% RSLogix 500 project STRAPPER 21-1-08 1220 - IN USE.RSS, saved by version 7.00.00.19 %
PROJECT "STRAPSYS"    % processor: MicroLogix 1500 %

PROGRAM FILES
  LAD 2 "MAIN"  17 rungs
  LAD 3 "INPUTS"  67 rungs
  LAD 4 "OUTPUTS"  55 rungs
  LAD 5 "INTERF OP"  16 rungs
  LAD 6 "COEFF."  16 rungs  % COEFFICIENT OF SEALING %
  LAD 7 "DISPENSER"  18 rungs
  LAD 8 "MH600"  137 rungs
  LAD 9 "ORGANIT."  67 rungs
  LAD 10 "PRESS"  78 rungs
  LAD 11 "PUSH_BUNK"  101 rungs
  LAD 12 "CHECKING"  10 rungs
  LAD 13 "INFEED"  25 rungs  % INFEED CONTROLS %
  LAD 14 "OUTFEED"  12 rungs  % OUTFEED CONTROLS %
  LAD 15 "RECIPES"  18 rungs  % PV RECIPE CONTROL %
  LAD 16 "ENCODER"  10 rungs  % ENCODER %
  LAD 17 "VSD"  10 rungs  % INFEED VSD'S %
  LAD 18 "RECIPE SEQ"  29 rungs

DATA FILES
  O0 OUTPUTS  9 elements
  I1 INPUT  10 elements
  S2 STATUS  66 elements
  B3 BINARY  30 elements
  T4 TIMER  52 elements
  C5 COUNTER  1 elements
  R6 CONTROL  1 elements
  N7 INTEGER  68 elements
  F8 FLOAT  9 elements
  N9 OP  13 elements
  B10 ORGANIT  106 elements
  N11 ON_SHOOT  3 elements
  L12   16 elements
  B20 MH600  101 elements
  B35 DISPENSER  9 elements
  B40 INFEEDBIN  100 elements  % INFEED SYSTEM BINARY %
  T41 INFEEDTIM  100 elements  % INFEED TIMERS %
  N42 INFEEDINT  100 elements  % INFEED INTEGERS %
  B50 PUSH_BUNK  24 elements
  N51 RECIPE  170 elements
  N52 REC NAMES  160 elements

LADDER 2 "MAIN"
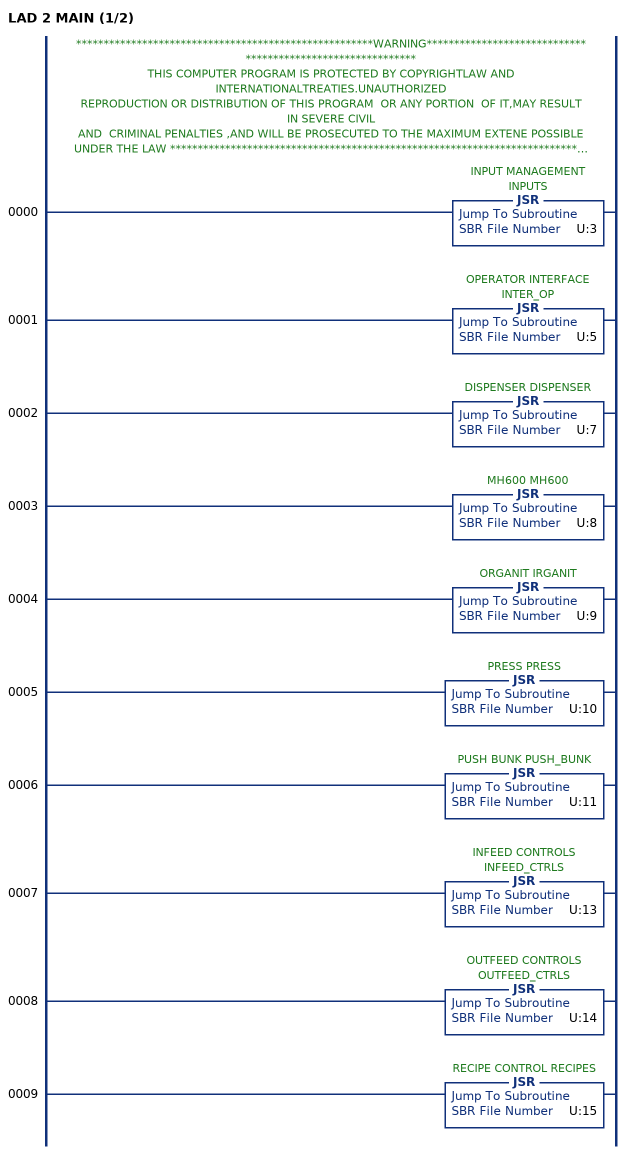
% Rung: 0 %
% ******************************************************WARNING************************************************************
% THIS COMPUTER PROGRAM IS PROTECTED BY COPYRIGHTLAW AND  INTERNATIONALTREATIES.UNAUTHORIZED
%  REPRODUCTION OR DISTRIBUTION OF THIS PROGRAM  OR ANY PORTION  OF IT,MAY RESULT IN SEVERE CIVIL
% AND  CRIMINAL PENALTIES ,AND WILL BE PROSECUTED TO THE MAXIMUM EXTENE POSSIBLE  UNDER THE LAW **************************************************************************************************************************
% Calls to the soubroutine %
SOR JSR U:3 EOR
%   U:3  INPUTS  "INPUT MANAGEMENT" %
% Rung: 1 %
SOR JSR U:5 EOR
%   U:5  INTER_OP  "OPERATOR INTERFACE" %
% Rung: 2 %
SOR JSR U:7 EOR
%   U:7  DISPENSER  "DISPENSER" %
% Rung: 3 %
SOR JSR U:8 EOR
%   U:8  MH600  "MH600" %
% Rung: 4 %
SOR JSR U:9 EOR
%   U:9  IRGANIT  "ORGANIT" %
% Rung: 5 %
SOR JSR U:10 EOR
%   U:10  PRESS  "PRESS" %
% Rung: 6 %
SOR JSR U:11 EOR
%   U:11  PUSH_BUNK  "PUSH BUNK" %
% Rung: 7 %
SOR JSR U:13 EOR
%   U:13  INFEED_CTRLS  "INFEED CONTROLS" %
% Rung: 8 %
SOR JSR U:14 EOR
%   U:14  OUTFEED_CTRLS  "OUTFEED CONTROLS" %
% Rung: 9 %
SOR JSR U:15 EOR
%   U:15  RECIPES  "RECIPE CONTROL" %

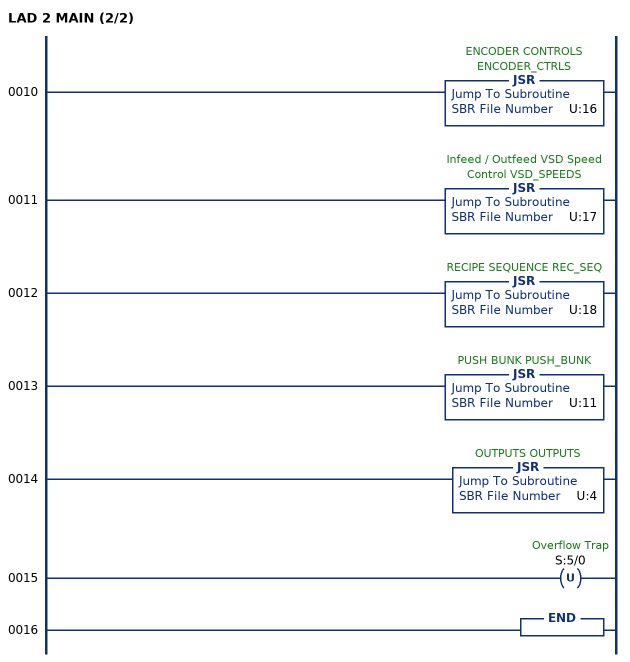
% Rung: 10 %
SOR JSR U:16 EOR
%   U:16  ENCODER_CTRLS  "ENCODER CONTROLS" %
% Rung: 11 %
SOR JSR U:17 EOR
%   U:17  VSD_SPEEDS  "Infeed / Outfeed VSD Speed Control" %
% Rung: 12 %
SOR JSR U:18 EOR
%   U:18  REC_SEQ  "RECIPE SEQUENCE" %
% Rung: 13 %
SOR JSR U:11 EOR
%   U:11  PUSH_BUNK  "PUSH BUNK" %
% Rung: 14 %
SOR JSR U:4 EOR
%   U:4  OUTPUTS  "OUTPUTS" %
% Rung: 15 %
SOR OTU S:5/0 EOR
%   S:5/0  "Overflow Trap" %
% Rung: 16 %
SOR END EOR

LADDER 3 "INPUTS"
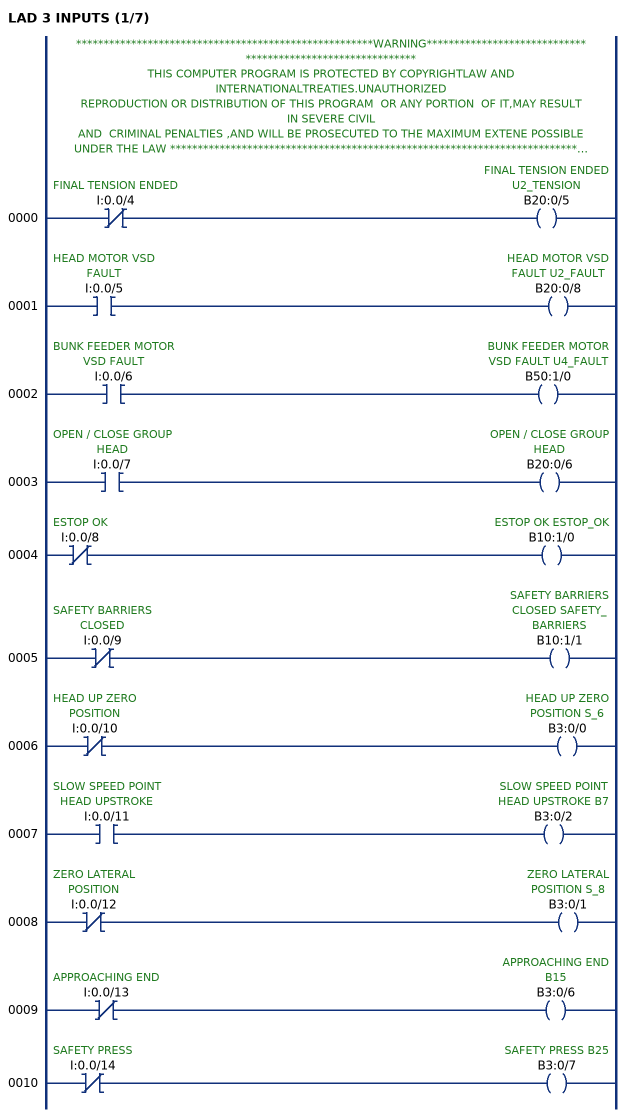
% Rung: 0 %
% ******************************************************WARNING************************************************************
% THIS COMPUTER PROGRAM IS PROTECTED BY COPYRIGHTLAW AND  INTERNATIONALTREATIES.UNAUTHORIZED
%  REPRODUCTION OR DISTRIBUTION OF THIS PROGRAM  OR ANY PORTION  OF IT,MAY RESULT IN SEVERE CIVIL
% AND  CRIMINAL PENALTIES ,AND WILL BE PROSECUTED TO THE MAXIMUM EXTENE POSSIBLE  UNDER THE LAW **************************************************************************************************************************
% AUTOMATIC VERTICAL PLASTIC MACHINE - I/O LOADING %
SOR XIO I:0.0/4 OTE B20:0/5 EOR
%   I:0.0/4  "FINAL TENSION ENDED" %
%   B20:0/5  U2_TENSION  "FINAL TENSION ENDED" %
% Rung: 1 %
SOR XIC I:0.0/5 OTE B20:0/8 EOR
%   I:0.0/5  "HEAD MOTOR VSD FAULT" %
%   B20:0/8  U2_FAULT  "HEAD MOTOR VSD FAULT" %
% Rung: 2 %
SOR XIC I:0.0/6 OTE B50:1/0 EOR
%   I:0.0/6  "BUNK FEEDER MOTOR VSD FAULT" %
%   B50:1/0  U4_FAULT  "BUNK FEEDER MOTOR VSD FAULT" %
% Rung: 3 %
SOR XIC I:0.0/7 OTE B20:0/6 EOR
%   I:0.0/7  "OPEN / CLOSE GROUP HEAD" %
%   B20:0/6  "OPEN / CLOSE GROUP HEAD" %
% Rung: 4 %
SOR XIO I:0.0/8 OTE B10:1/0 EOR
%   I:0.0/8  "ESTOP OK" %
%   B10:1/0  ESTOP_OK  "ESTOP OK" %
% Rung: 5 %
SOR XIO I:0.0/9 OTE B10:1/1 EOR
%   I:0.0/9  "SAFETY BARRIERS CLOSED" %
%   B10:1/1  SAFETY_BARRIERS  "SAFETY BARRIERS CLOSED" %
% Rung: 6 %
SOR XIO I:0.0/10 OTE B3:0/0 EOR
%   I:0.0/10  "HEAD UP ZERO POSITION" %
%   B3:0/0  S_6  "HEAD UP ZERO POSITION" %
% Rung: 7 %
SOR XIC I:0.0/11 OTE B3:0/2 EOR
%   I:0.0/11  "SLOW SPEED POINT HEAD UPSTROKE" %
%   B3:0/2  B7  "SLOW SPEED POINT HEAD UPSTROKE" %
% Rung: 8 %
SOR XIO I:0.0/12 OTE B3:0/1 EOR
%   I:0.0/12  "ZERO LATERAL POSITION" %
%   B3:0/1  S_8  "ZERO LATERAL POSITION" %
% Rung: 9 %
SOR XIO I:0.0/13 OTE B3:0/6 EOR
%   I:0.0/13  "APPROACHING END" %
%   B3:0/6  B15  "APPROACHING END" %
% Rung: 10 %
SOR XIO I:0.0/14 OTE B3:0/7 EOR
%   I:0.0/14  "SAFETY PRESS" %
%   B3:0/7  B25  "SAFETY PRESS" %

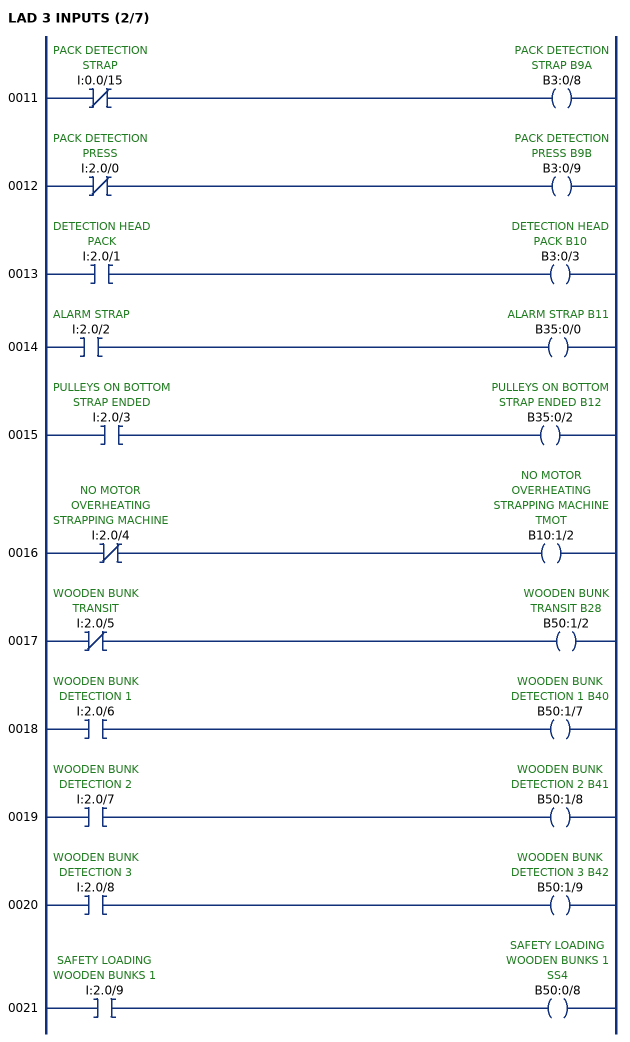
% Rung: 11 %
SOR XIO I:0.0/15 OTE B3:0/8 EOR
%   I:0.0/15  "PACK DETECTION STRAP" %
%   B3:0/8  B9A  "PACK DETECTION STRAP" %
% Rung: 12 %
SOR XIO I:2.0/0 OTE B3:0/9 EOR
%   I:2.0/0  "PACK DETECTION PRESS" %
%   B3:0/9  B9B  "PACK DETECTION PRESS" %
% Rung: 13 %
SOR XIC I:2.0/1 OTE B3:0/3 EOR
%   I:2.0/1  "DETECTION HEAD PACK" %
%   B3:0/3  B10  "DETECTION HEAD PACK" %
% Rung: 14 %
SOR XIC I:2.0/2 OTE B35:0/0 EOR
%   I:2.0/2  "ALARM STRAP" %
%   B35:0/0  B11  "ALARM STRAP" %
% Rung: 15 %
SOR XIC I:2.0/3 OTE B35:0/2 EOR
%   I:2.0/3  "PULLEYS ON BOTTOM STRAP ENDED" %
%   B35:0/2  B12  "PULLEYS ON BOTTOM STRAP ENDED" %
% Rung: 16 %
SOR XIO I:2.0/4 OTE B10:1/2 EOR
%   I:2.0/4  "NO MOTOR OVERHEATING STRAPPING MACHINE" %
%   B10:1/2  TMOT  "NO MOTOR OVERHEATING STRAPPING MACHINE" %
% Rung: 17 %
SOR XIO I:2.0/5 OTE B50:1/2 EOR
%   I:2.0/5  "WOODEN BUNK TRANSIT" %
%   B50:1/2  B28  "WOODEN BUNK TRANSIT" %
% Rung: 18 %
SOR XIC I:2.0/6 OTE B50:1/7 EOR
%   I:2.0/6  "WOODEN BUNK DETECTION 1" %
%   B50:1/7  B40  "WOODEN BUNK DETECTION 1" %
% Rung: 19 %
SOR XIC I:2.0/7 OTE B50:1/8 EOR
%   I:2.0/7  "WOODEN BUNK DETECTION 2" %
%   B50:1/8  B41  "WOODEN BUNK DETECTION 2" %
% Rung: 20 %
SOR XIC I:2.0/8 OTE B50:1/9 EOR
%   I:2.0/8  "WOODEN BUNK DETECTION 3" %
%   B50:1/9  B42  "WOODEN BUNK DETECTION 3" %
% Rung: 21 %
SOR XIC I:2.0/9 OTE B50:0/8 EOR
%   I:2.0/9  "SAFETY LOADING WOODEN BUNKS 1" %
%   B50:0/8  SS4  "SAFETY LOADING WOODEN BUNKS 1" %

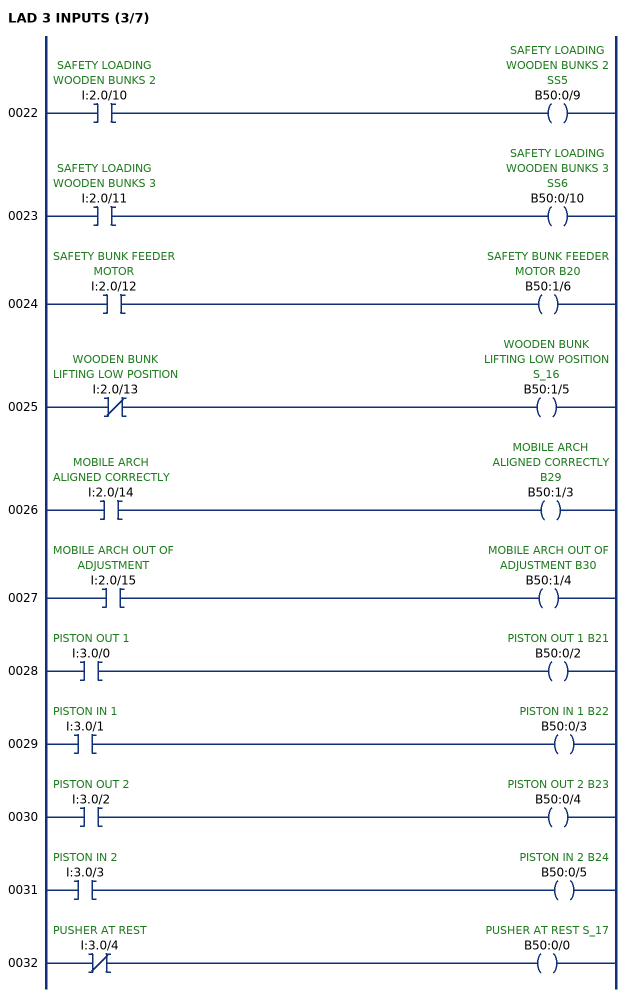
% Rung: 22 %
SOR XIC I:2.0/10 OTE B50:0/9 EOR
%   I:2.0/10  "SAFETY LOADING WOODEN BUNKS 2" %
%   B50:0/9  SS5  "SAFETY LOADING WOODEN BUNKS 2" %
% Rung: 23 %
SOR XIC I:2.0/11 OTE B50:0/10 EOR
%   I:2.0/11  "SAFETY LOADING WOODEN BUNKS 3" %
%   B50:0/10  SS6  "SAFETY LOADING WOODEN BUNKS 3" %
% Rung: 24 %
SOR XIC I:2.0/12 OTE B50:1/6 EOR
%   I:2.0/12  "SAFETY BUNK FEEDER MOTOR" %
%   B50:1/6  B20  "SAFETY BUNK FEEDER MOTOR" %
% Rung: 25 %
SOR XIO I:2.0/13 OTE B50:1/5 EOR
%   I:2.0/13  "WOODEN BUNK LIFTING LOW POSITION" %
%   B50:1/5  S_16  "WOODEN BUNK LIFTING LOW POSITION" %
% Rung: 26 %
SOR XIC I:2.0/14 OTE B50:1/3 EOR
%   I:2.0/14  "MOBILE ARCH ALIGNED CORRECTLY" %
%   B50:1/3  B29  "MOBILE ARCH ALIGNED CORRECTLY" %
% Rung: 27 %
SOR XIC I:2.0/15 OTE B50:1/4 EOR
%   I:2.0/15  "MOBILE ARCH OUT OF ADJUSTMENT" %
%   B50:1/4  B30  "MOBILE ARCH OUT OF ADJUSTMENT" %
% Rung: 28 %
SOR XIC I:3.0/0 OTE B50:0/2 EOR
%   I:3.0/0  "PISTON OUT 1" %
%   B50:0/2  B21  "PISTON OUT 1" %
% Rung: 29 %
SOR XIC I:3.0/1 OTE B50:0/3 EOR
%   I:3.0/1  "PISTON IN 1" %
%   B50:0/3  B22  "PISTON IN 1" %
% Rung: 30 %
SOR XIC I:3.0/2 OTE B50:0/4 EOR
%   I:3.0/2  "PISTON OUT 2" %
%   B50:0/4  B23  "PISTON OUT 2" %
% Rung: 31 %
SOR XIC I:3.0/3 OTE B50:0/5 EOR
%   I:3.0/3  "PISTON IN 2" %
%   B50:0/5  B24  "PISTON IN 2" %
% Rung: 32 %
SOR XIO I:3.0/4 OTE B50:0/0 EOR
%   I:3.0/4  "PUSHER AT REST" %
%   B50:0/0  S_17  "PUSHER AT REST" %

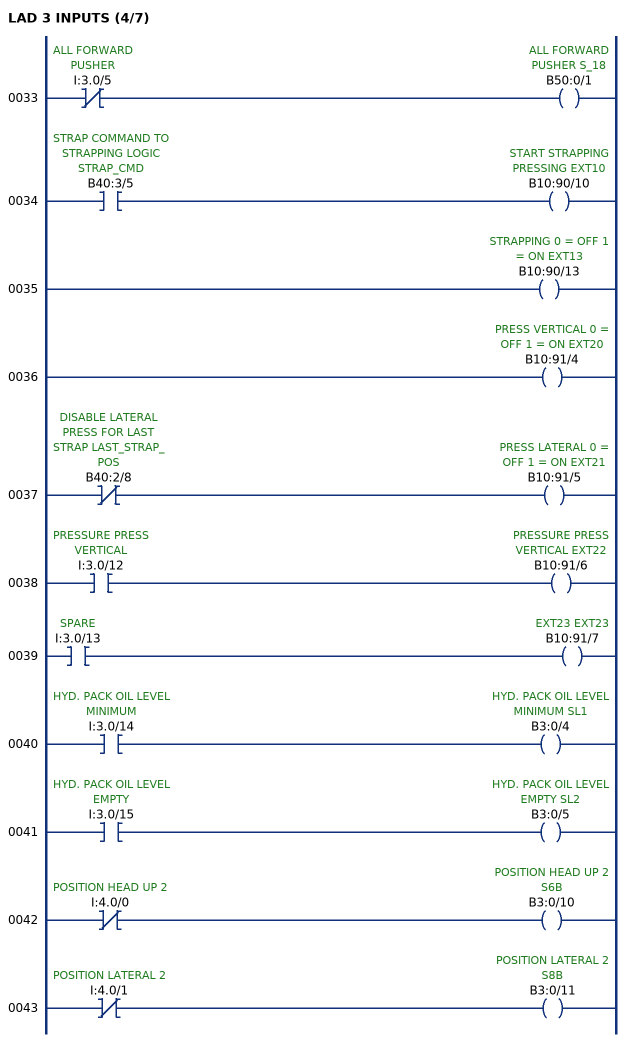
% Rung: 33 %
SOR XIO I:3.0/5 OTE B50:0/1 EOR
%   I:3.0/5  "ALL FORWARD PUSHER" %
%   B50:0/1  S_18  "ALL FORWARD PUSHER" %
% Rung: 34 %
SOR XIC B40:3/5 OTE B10:90/10 EOR
%   B40:3/5  STRAP_CMD  "STRAP COMMAND TO STRAPPING LOGIC" %
%   B10:90/10  EXT10  "START STRAPPING PRESSING" %
% Rung: 35 %
SOR OTE B10:90/13 EOR
%   B10:90/13  EXT13  "STRAPPING 0 = OFF 1 = ON" %
% Rung: 36 %
SOR OTE B10:91/4 EOR
%   B10:91/4  EXT20  "PRESS VERTICAL 0 = OFF 1 = ON" %
% Rung: 37 %
SOR XIO B40:2/8 OTE B10:91/5 EOR
%   B40:2/8  LAST_STRAP_POS  "DISABLE LATERAL PRESS FOR LAST STRAP" %
%   B10:91/5  EXT21  "PRESS LATERAL 0 = OFF 1 = ON" %
% Rung: 38 %
SOR XIC I:3.0/12 OTE B10:91/6 EOR
%   I:3.0/12  "PRESSURE PRESS VERTICAL" %
%   B10:91/6  EXT22  "PRESSURE PRESS VERTICAL" %
% Rung: 39 %
SOR XIC I:3.0/13 OTE B10:91/7 EOR
%   I:3.0/13  "SPARE" %
%   B10:91/7  EXT23  "EXT23" %
% Rung: 40 %
SOR XIC I:3.0/14 OTE B3:0/4 EOR
%   I:3.0/14  "HYD. PACK OIL LEVEL MINIMUM" %
%   B3:0/4  SL1  "HYD. PACK OIL LEVEL MINIMUM" %
% Rung: 41 %
SOR XIC I:3.0/15 OTE B3:0/5 EOR
%   I:3.0/15  "HYD. PACK OIL LEVEL EMPTY" %
%   B3:0/5  SL2  "HYD. PACK OIL LEVEL EMPTY" %
% Rung: 42 %
SOR XIO I:4.0/0 OTE B3:0/10 EOR
%   I:4.0/0  "POSITION HEAD UP 2" %
%   B3:0/10  S6B  "POSITION HEAD UP 2" %
% Rung: 43 %
SOR XIO I:4.0/1 OTE B3:0/11 EOR
%   I:4.0/1  "POSITION LATERAL 2" %
%   B3:0/11  S8B  "POSITION LATERAL 2" %

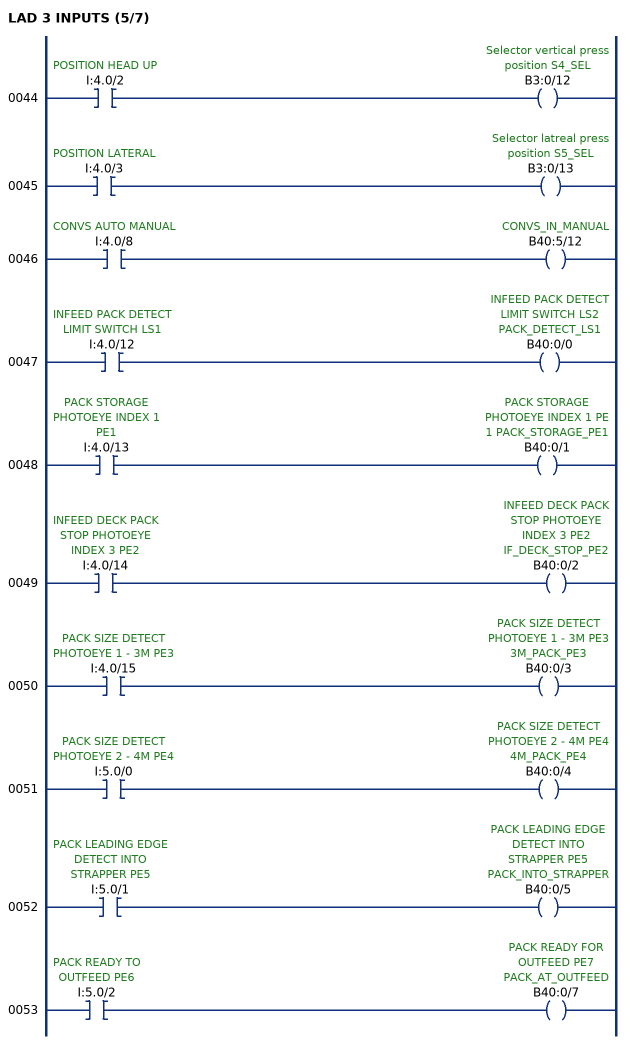
% Rung: 44 %
SOR XIC I:4.0/2 OTE B3:0/12 EOR
%   I:4.0/2  "POSITION HEAD UP" %
%   B3:0/12  S4_SEL  "Selector vertical press position" %
% Rung: 45 %
SOR XIC I:4.0/3 OTE B3:0/13 EOR
%   I:4.0/3  "POSITION LATERAL" %
%   B3:0/13  S5_SEL  "Selector latreal press position" %
% Rung: 46 %
SOR XIC I:4.0/8 OTE B40:5/12 EOR
%   I:4.0/8  "CONVS AUTO MANUAL" %
%   B40:5/12  CONVS_IN_MANUAL %
% Rung: 47 %
SOR XIC I:4.0/12 OTE B40:0/0 EOR
%   I:4.0/12  "INFEED PACK DETECT LIMIT SWITCH LS1" %
%   B40:0/0  PACK_DETECT_LS1  "INFEED PACK DETECT LIMIT SWITCH LS2" %
% Rung: 48 %
SOR XIC I:4.0/13 OTE B40:0/1 EOR
%   I:4.0/13  "PACK STORAGE PHOTOEYE INDEX 1 PE1" %
%   B40:0/1  PACK_STORAGE_PE1  "PACK STORAGE PHOTOEYE INDEX 1 PE 1" %
% Rung: 49 %
SOR XIC I:4.0/14 OTE B40:0/2 EOR
%   I:4.0/14  "INFEED DECK PACK STOP PHOTOEYE INDEX 3 PE2" %
%   B40:0/2  IF_DECK_STOP_PE2  "INFEED DECK PACK STOP PHOTOEYE INDEX 3 PE2" %
% Rung: 50 %
SOR XIC I:4.0/15 OTE B40:0/3 EOR
%   I:4.0/15  "PACK SIZE DETECT PHOTOEYE 1 - 3M PE3" %
%   B40:0/3  3M_PACK_PE3  "PACK SIZE DETECT PHOTOEYE 1 - 3M PE3" %
% Rung: 51 %
SOR XIC I:5.0/0 OTE B40:0/4 EOR
%   I:5.0/0  "PACK SIZE DETECT PHOTOEYE 2 - 4M PE4" %
%   B40:0/4  4M_PACK_PE4  "PACK SIZE DETECT PHOTOEYE 2 - 4M PE4" %
% Rung: 52 %
SOR XIC I:5.0/1 OTE B40:0/5 EOR
%   I:5.0/1  "PACK LEADING EDGE DETECT INTO STRAPPER PE5" %
%   B40:0/5  PACK_INTO_STRAPPER  "PACK LEADING EDGE DETECT INTO STRAPPER PE5" %
% Rung: 53 %
SOR XIC I:5.0/2 OTE B40:0/7 EOR
%   I:5.0/2  "PACK READY TO OUTFEED PE6" %
%   B40:0/7  PACK_AT_OUTFEED  "PACK READY FOR OUTFEED PE7" %

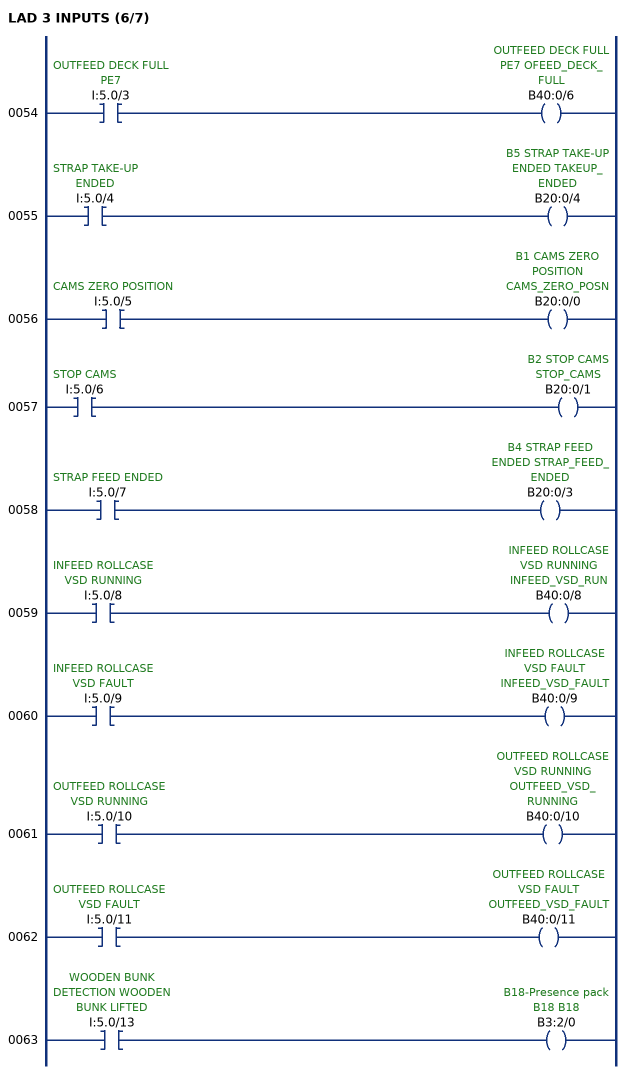
% Rung: 54 %
SOR XIC I:5.0/3 OTE B40:0/6 EOR
%   I:5.0/3  "OUTFEED DECK FULL PE7" %
%   B40:0/6  OFEED_DECK_FULL  "OUTFEED DECK FULL PE7" %
% Rung: 55 %
SOR XIC I:5.0/4 OTE B20:0/4 EOR
%   I:5.0/4  "STRAP TAKE-UP ENDED" %
%   B20:0/4  TAKEUP_ENDED  "B5 STRAP TAKE-UP ENDED" %
% Rung: 56 %
SOR XIC I:5.0/5 OTE B20:0/0 EOR
%   I:5.0/5  "CAMS ZERO POSITION" %
%   B20:0/0  CAMS_ZERO_POSN  "B1 CAMS ZERO POSITION" %
% Rung: 57 %
SOR XIC I:5.0/6 OTE B20:0/1 EOR
%   I:5.0/6  "STOP CAMS" %
%   B20:0/1  STOP_CAMS  "B2 STOP CAMS" %
% Rung: 58 %
SOR XIC I:5.0/7 OTE B20:0/3 EOR
%   I:5.0/7  "STRAP FEED ENDED" %
%   B20:0/3  STRAP_FEED_ENDED  "B4 STRAP FEED ENDED" %
% Rung: 59 %
SOR XIC I:5.0/8 OTE B40:0/8 EOR
%   I:5.0/8  "INFEED ROLLCASE VSD RUNNING" %
%   B40:0/8  INFEED_VSD_RUN  "INFEED ROLLCASE VSD RUNNING" %
% Rung: 60 %
SOR XIC I:5.0/9 OTE B40:0/9 EOR
%   I:5.0/9  "INFEED ROLLCASE VSD FAULT" %
%   B40:0/9  INFEED_VSD_FAULT  "INFEED ROLLCASE VSD FAULT" %
% Rung: 61 %
SOR XIC I:5.0/10 OTE B40:0/10 EOR
%   I:5.0/10  "OUTFEED ROLLCASE VSD RUNNING" %
%   B40:0/10  OUTFEED_VSD_RUNNING  "OUTFEED ROLLCASE VSD RUNNING" %
% Rung: 62 %
SOR XIC I:5.0/11 OTE B40:0/11 EOR
%   I:5.0/11  "OUTFEED ROLLCASE VSD FAULT" %
%   B40:0/11  OUTFEED_VSD_FAULT  "OUTFEED ROLLCASE VSD FAULT" %
% Rung: 63 %
SOR XIC I:5.0/13 OTE B3:2/0 EOR
%   I:5.0/13  "WOODEN BUNK DETECTION WOODEN BUNK LIFTED" %
%   B3:2/0  B18  "B18-Presence pack B18" %

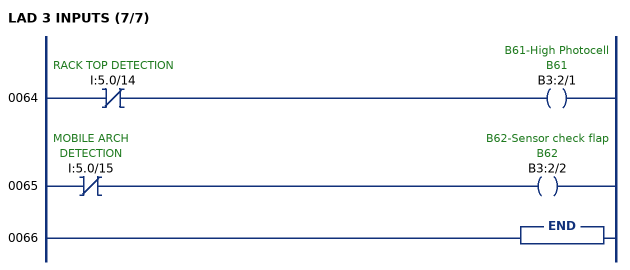
% Rung: 64 %
SOR XIO I:5.0/14 OTE B3:2/1 EOR
%   I:5.0/14  "RACK TOP DETECTION" %
%   B3:2/1  B61  "B61-High Photocell" %
% Rung: 65 %
SOR XIO I:5.0/15 OTE B3:2/2 EOR
%   I:5.0/15  "MOBILE ARCH DETECTION" %
%   B3:2/2  B62  "B62-Sensor check flap" %
% Rung: 66 %
SOR END EOR

LADDER 4 "OUTPUTS"
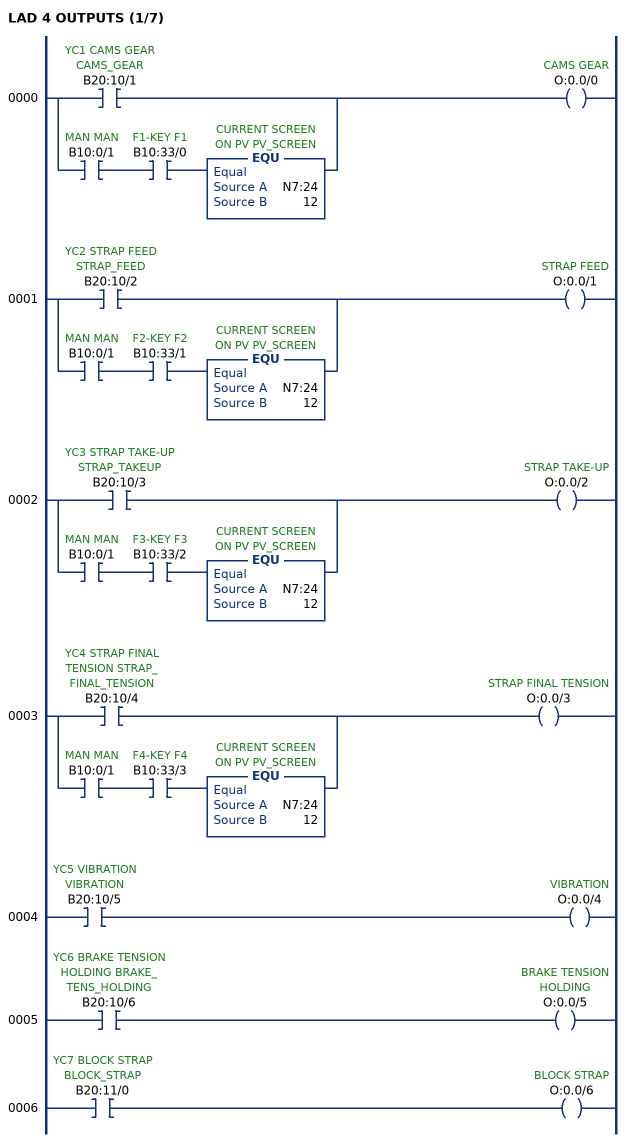
% Rung: 0 %
SOR BST XIC B20:10/1 NXB XIC B10:0/1 XIC B10:33/0 EQU N7:24 12 BND OTE O:0.0/0 EOR
%   B20:10/1  CAMS_GEAR  "YC1 CAMS GEAR" %
%   B10:0/1  MAN  "MAN" %
%   B10:33/0  F1  "F1-KEY" %
%   N7:24  PV_SCREEN  "CURRENT SCREEN ON PV" %
%   O:0.0/0  "CAMS GEAR" %
% Rung: 1 %
SOR BST XIC B20:10/2 NXB XIC B10:0/1 XIC B10:33/1 EQU N7:24 12 BND OTE O:0.0/1 EOR
%   B20:10/2  STRAP_FEED  "YC2 STRAP FEED" %
%   B10:0/1  MAN  "MAN" %
%   B10:33/1  F2  "F2-KEY" %
%   N7:24  PV_SCREEN  "CURRENT SCREEN ON PV" %
%   O:0.0/1  "STRAP FEED" %
% Rung: 2 %
SOR BST XIC B20:10/3 NXB XIC B10:0/1 XIC B10:33/2 EQU N7:24 12 BND OTE O:0.0/2 EOR
%   B20:10/3  STRAP_TAKEUP  "YC3 STRAP TAKE-UP" %
%   B10:0/1  MAN  "MAN" %
%   B10:33/2  F3  "F3-KEY" %
%   N7:24  PV_SCREEN  "CURRENT SCREEN ON PV" %
%   O:0.0/2  "STRAP TAKE-UP" %
% Rung: 3 %
SOR BST XIC B20:10/4 NXB XIC B10:0/1 XIC B10:33/3 EQU N7:24 12 BND OTE O:0.0/3 EOR
%   B20:10/4  STRAP_FINAL_TENSION  "YC4 STRAP FINAL TENSION" %
%   B10:0/1  MAN  "MAN" %
%   B10:33/3  F4  "F4-KEY" %
%   N7:24  PV_SCREEN  "CURRENT SCREEN ON PV" %
%   O:0.0/3  "STRAP FINAL TENSION" %
% Rung: 4 %
SOR XIC B20:10/5 OTE O:0.0/4 EOR
%   B20:10/5  VIBRATION  "YC5 VIBRATION" %
%   O:0.0/4  "VIBRATION" %
% Rung: 5 %
SOR XIC B20:10/6 OTE O:0.0/5 EOR
%   B20:10/6  BRAKE_TENS_HOLDING  "YC6 BRAKE TENSION HOLDING" %
%   O:0.0/5  "BRAKE TENSION HOLDING" %
% Rung: 6 %
SOR XIC B20:11/0 OTE O:0.0/6 EOR
%   B20:11/0  BLOCK_STRAP  "YC7 BLOCK STRAP" %
%   O:0.0/6  "BLOCK STRAP" %

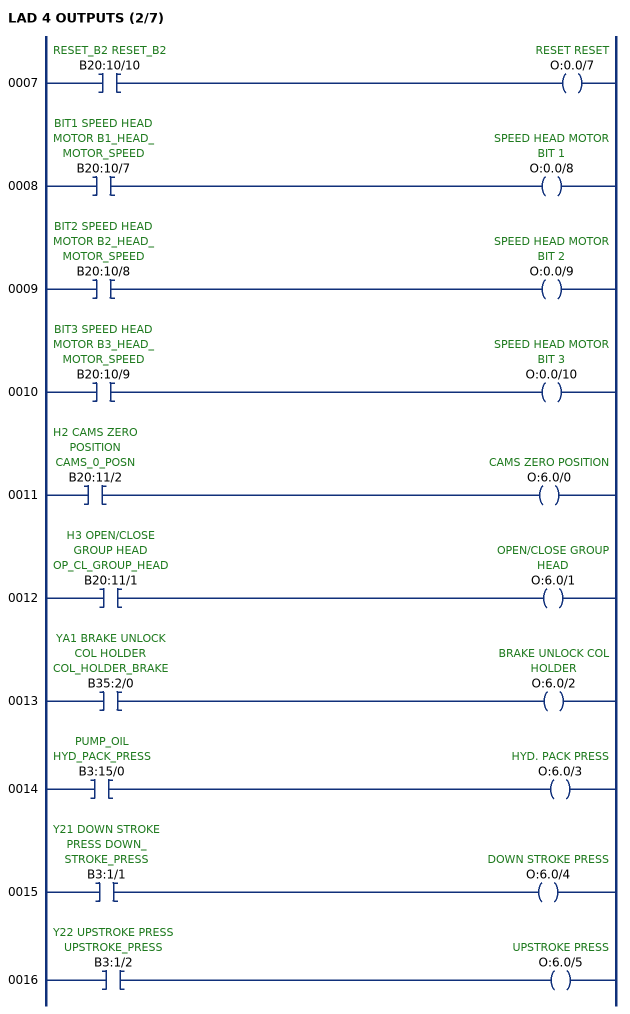
% Rung: 7 %
SOR XIC B20:10/10 OTE O:0.0/7 EOR
%   B20:10/10  RESET_B2  "RESET_B2" %
%   O:0.0/7  RESET  "RESET" %
% Rung: 8 %
SOR XIC B20:10/7 OTE O:0.0/8 EOR
%   B20:10/7  B1_HEAD_MOTOR_SPEED  "BIT1 SPEED HEAD MOTOR" %
%   O:0.0/8  "SPEED HEAD MOTOR BIT 1" %
% Rung: 9 %
SOR XIC B20:10/8 OTE O:0.0/9 EOR
%   B20:10/8  B2_HEAD_MOTOR_SPEED  "BIT2 SPEED HEAD MOTOR" %
%   O:0.0/9  "SPEED HEAD MOTOR BIT 2" %
% Rung: 10 %
SOR XIC B20:10/9 OTE O:0.0/10 EOR
%   B20:10/9  B3_HEAD_MOTOR_SPEED  "BIT3 SPEED HEAD MOTOR" %
%   O:0.0/10  "SPEED HEAD MOTOR BIT 3" %
% Rung: 11 %
SOR XIC B20:11/2 OTE O:6.0/0 EOR
%   B20:11/2  CAMS_0_POSN  "H2 CAMS ZERO POSITION" %
%   O:6.0/0  "CAMS ZERO POSITION" %
% Rung: 12 %
SOR XIC B20:11/1 OTE O:6.0/1 EOR
%   B20:11/1  OP_CL_GROUP_HEAD  "H3 OPEN/CLOSE GROUP HEAD" %
%   O:6.0/1  "OPEN/CLOSE GROUP HEAD" %
% Rung: 13 %
SOR XIC B35:2/0 OTE O:6.0/2 EOR
%   B35:2/0  COL_HOLDER_BRAKE  "YA1 BRAKE UNLOCK COL HOLDER" %
%   O:6.0/2  "BRAKE UNLOCK COL HOLDER" %
% Rung: 14 %
SOR XIC B3:15/0 OTE O:6.0/3 EOR
%   B3:15/0  HYD_PACK_PRESS  "PUMP_OIL" %
%   O:6.0/3  "HYD. PACK PRESS" %
% Rung: 15 %
SOR XIC B3:1/1 OTE O:6.0/4 EOR
%   B3:1/1  DOWN_STROKE_PRESS  "Y21 DOWN STROKE PRESS" %
%   O:6.0/4  "DOWN STROKE PRESS" %
% Rung: 16 %
SOR XIC B3:1/2 OTE O:6.0/5 EOR
%   B3:1/2  UPSTROKE_PRESS  "Y22 UPSTROKE PRESS" %
%   O:6.0/5  "UPSTROKE PRESS" %

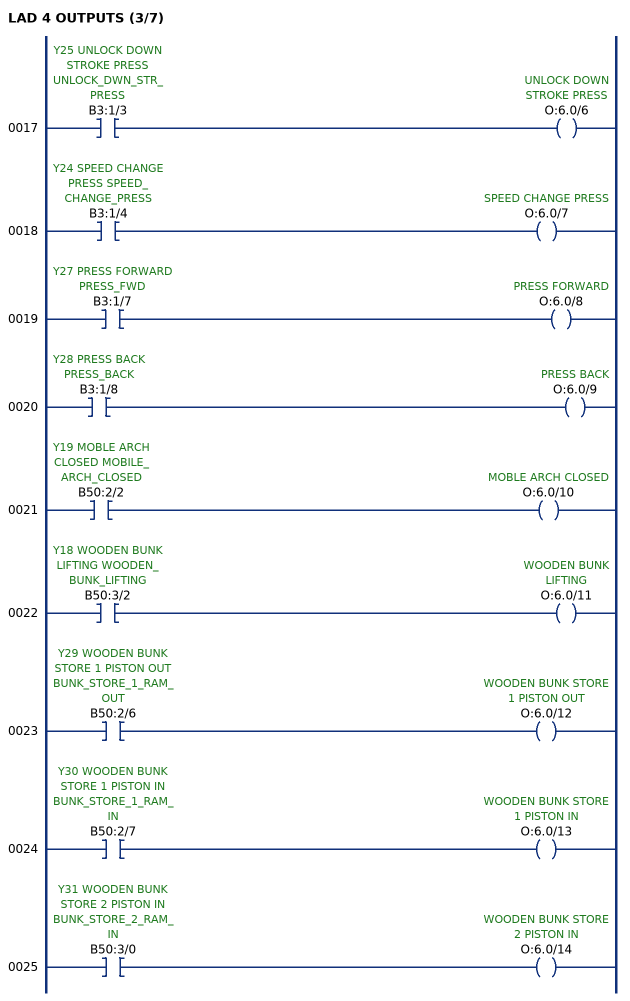
% Rung: 17 %
SOR XIC B3:1/3 OTE O:6.0/6 EOR
%   B3:1/3  UNLOCK_DWN_STR_PRESS  "Y25 UNLOCK DOWN STROKE PRESS" %
%   O:6.0/6  "UNLOCK DOWN STROKE PRESS" %
% Rung: 18 %
SOR XIC B3:1/4 OTE O:6.0/7 EOR
%   B3:1/4  SPEED_CHANGE_PRESS  "Y24 SPEED CHANGE PRESS" %
%   O:6.0/7  "SPEED CHANGE PRESS" %
% Rung: 19 %
SOR XIC B3:1/7 OTE O:6.0/8 EOR
%   B3:1/7  PRESS_FWD  "Y27 PRESS FORWARD" %
%   O:6.0/8  "PRESS FORWARD" %
% Rung: 20 %
SOR XIC B3:1/8 OTE O:6.0/9 EOR
%   B3:1/8  PRESS_BACK  "Y28 PRESS BACK" %
%   O:6.0/9  "PRESS BACK" %
% Rung: 21 %
SOR XIC B50:2/2 OTE O:6.0/10 EOR
%   B50:2/2  MOBILE_ARCH_CLOSED  "Y19 MOBLE ARCH CLOSED" %
%   O:6.0/10  "MOBLE ARCH CLOSED" %
% Rung: 22 %
SOR XIC B50:3/2 OTE O:6.0/11 EOR
%   B50:3/2  WOODEN_BUNK_LIFTING  "Y18 WOODEN BUNK LIFTING" %
%   O:6.0/11  "WOODEN BUNK LIFTING" %
% Rung: 23 %
SOR XIC B50:2/6 OTE O:6.0/12 EOR
%   B50:2/6  BUNK_STORE_1_RAM_OUT  "Y29 WOODEN BUNK STORE 1 PISTON OUT" %
%   O:6.0/12  "WOODEN BUNK STORE 1 PISTON OUT" %
% Rung: 24 %
SOR XIC B50:2/7 OTE O:6.0/13 EOR
%   B50:2/7  BUNK_STORE_1_RAM_IN  "Y30 WOODEN BUNK STORE 1 PISTON IN" %
%   O:6.0/13  "WOODEN BUNK STORE 1 PISTON IN" %
% Rung: 25 %
SOR XIC B50:3/0 OTE O:6.0/14 EOR
%   B50:3/0  BUNK_STORE_2_RAM_IN  "Y31 WOODEN BUNK STORE 2 PISTON IN" %
%   O:6.0/14  "WOODEN BUNK STORE 2 PISTON IN" %

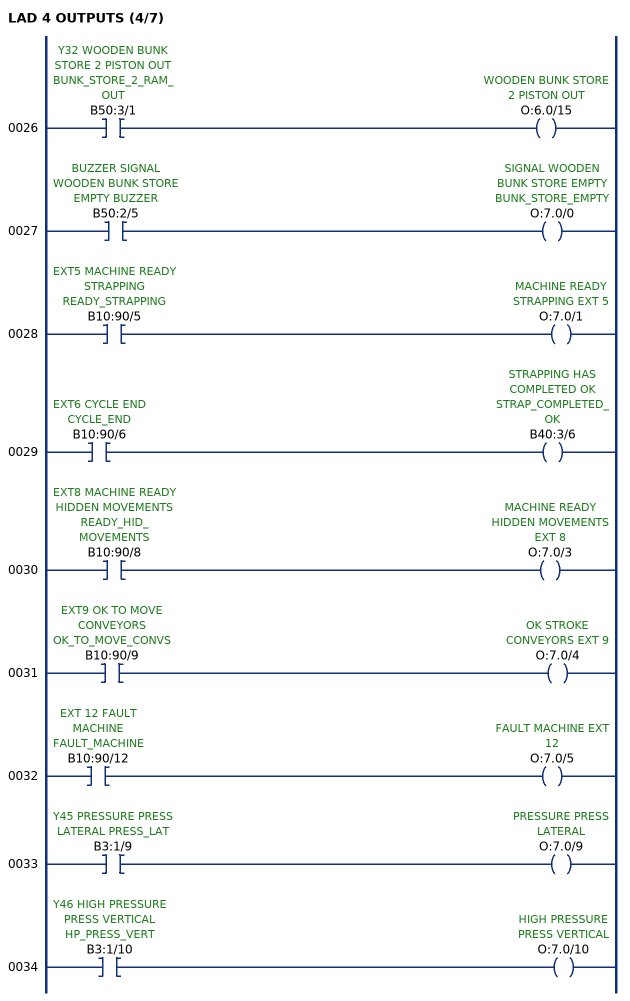
% Rung: 26 %
SOR XIC B50:3/1 OTE O:6.0/15 EOR
%   B50:3/1  BUNK_STORE_2_RAM_OUT  "Y32 WOODEN BUNK STORE 2 PISTON OUT" %
%   O:6.0/15  "WOODEN BUNK STORE 2 PISTON OUT" %
% Rung: 27 %
SOR XIC B50:2/5 OTE O:7.0/0 EOR
%   B50:2/5  BUZZER  "BUZZER SIGNAL WOODEN BUNK STORE EMPTY" %
%   O:7.0/0  BUNK_STORE_EMPTY  "SIGNAL WOODEN BUNK STORE EMPTY" %
% Rung: 28 %
SOR XIC B10:90/5 OTE O:7.0/1 EOR
%   B10:90/5  READY_STRAPPING  "EXT5 MACHINE READY STRAPPING" %
%   O:7.0/1  "MACHINE READY STRAPPING EXT 5" %
% Rung: 29 %
SOR XIC B10:90/6 OTE B40:3/6 EOR
%   B10:90/6  CYCLE_END  "EXT6 CYCLE END" %
%   B40:3/6  STRAP_COMPLETED_OK  "STRAPPING HAS COMPLETED OK" %
% Rung: 30 %
SOR XIC B10:90/8 OTE O:7.0/3 EOR
%   B10:90/8  READY_HID_MOVEMENTS  "EXT8 MACHINE READY HIDDEN MOVEMENTS" %
%   O:7.0/3  "MACHINE READY HIDDEN MOVEMENTS EXT 8" %
% Rung: 31 %
SOR XIC B10:90/9 OTE O:7.0/4 EOR
%   B10:90/9  OK_TO_MOVE_CONVS  "EXT9 OK TO MOVE CONVEYORS" %
%   O:7.0/4  "OK STROKE CONVEYORS EXT 9" %
% Rung: 32 %
SOR XIC B10:90/12 OTE O:7.0/5 EOR
%   B10:90/12  FAULT_MACHINE  "EXT 12 FAULT MACHINE" %
%   O:7.0/5  "FAULT MACHINE EXT 12" %
% Rung: 33 %
SOR XIC B3:1/9 OTE O:7.0/9 EOR
%   B3:1/9  PRESS_LAT  "Y45 PRESSURE PRESS LATERAL" %
%   O:7.0/9  "PRESSURE PRESS LATERAL" %
% Rung: 34 %
SOR XIC B3:1/10 OTE O:7.0/10 EOR
%   B3:1/10  HP_PRESS_VERT  "Y46 HIGH PRESSURE PRESS VERTICAL" %
%   O:7.0/10  "HIGH PRESSURE PRESS VERTICAL" %

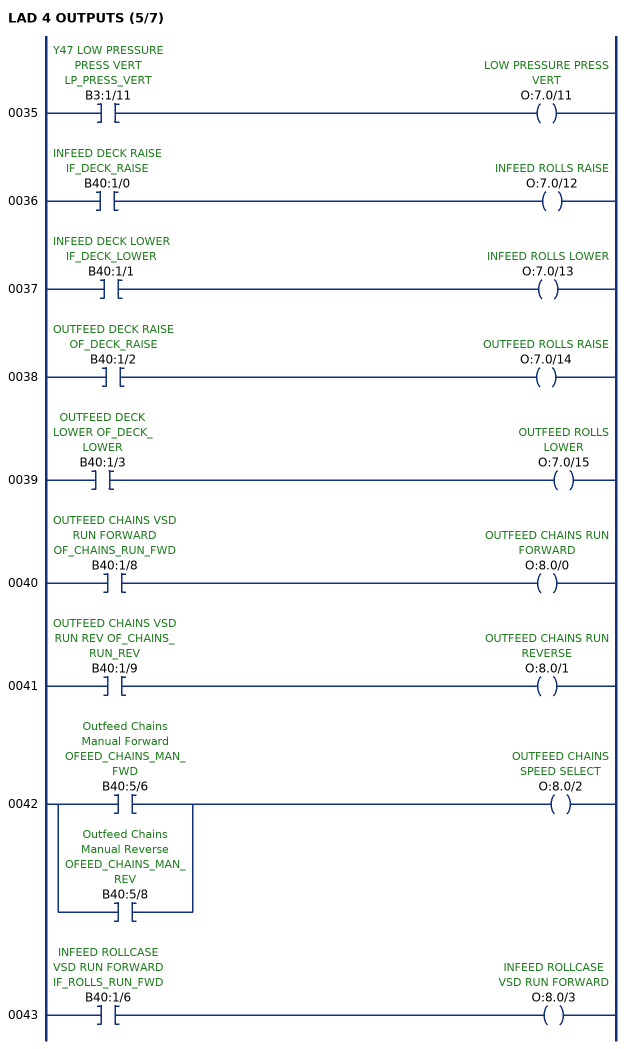
% Rung: 35 %
SOR XIC B3:1/11 OTE O:7.0/11 EOR
%   B3:1/11  LP_PRESS_VERT  "Y47 LOW PRESSURE PRESS VERT" %
%   O:7.0/11  "LOW PRESSURE PRESS VERT" %
% Rung: 36 %
SOR XIC B40:1/0 OTE O:7.0/12 EOR
%   B40:1/0  IF_DECK_RAISE  "INFEED DECK RAISE" %
%   O:7.0/12  "INFEED ROLLS RAISE" %
% Rung: 37 %
SOR XIC B40:1/1 OTE O:7.0/13 EOR
%   B40:1/1  IF_DECK_LOWER  "INFEED DECK LOWER" %
%   O:7.0/13  "INFEED ROLLS LOWER" %
% Rung: 38 %
SOR XIC B40:1/2 OTE O:7.0/14 EOR
%   B40:1/2  OF_DECK_RAISE  "OUTFEED DECK RAISE" %
%   O:7.0/14  "OUTFEED ROLLS RAISE" %
% Rung: 39 %
SOR XIC B40:1/3 OTE O:7.0/15 EOR
%   B40:1/3  OF_DECK_LOWER  "OUTFEED DECK LOWER" %
%   O:7.0/15  "OUTFEED ROLLS LOWER" %
% Rung: 40 %
SOR XIC B40:1/8 OTE O:8.0/0 EOR
%   B40:1/8  OF_CHAINS_RUN_FWD  "OUTFEED CHAINS VSD RUN FORWARD" %
%   O:8.0/0  "OUTFEED CHAINS RUN FORWARD" %
% Rung: 41 %
SOR XIC B40:1/9 OTE O:8.0/1 EOR
%   B40:1/9  OF_CHAINS_RUN_REV  "OUTFEED CHAINS VSD RUN REV" %
%   O:8.0/1  "OUTFEED CHAINS RUN REVERSE" %
% Rung: 42 %
SOR BST XIC B40:5/6 NXB XIC B40:5/8 BND OTE O:8.0/2 EOR
%   B40:5/6  OFEED_CHAINS_MAN_FWD  "Outfeed Chains Manual Forward" %
%   B40:5/8  OFEED_CHAINS_MAN_REV  "Outfeed Chains Manual Reverse" %
%   O:8.0/2  "OUTFEED CHAINS SPEED SELECT" %
% Rung: 43 %
SOR XIC B40:1/6 OTE O:8.0/3 EOR
%   B40:1/6  IF_ROLLS_RUN_FWD  "INFEED ROLLCASE VSD RUN FORWARD" %
%   O:8.0/3  "INFEED ROLLCASE VSD RUN FORWARD" %

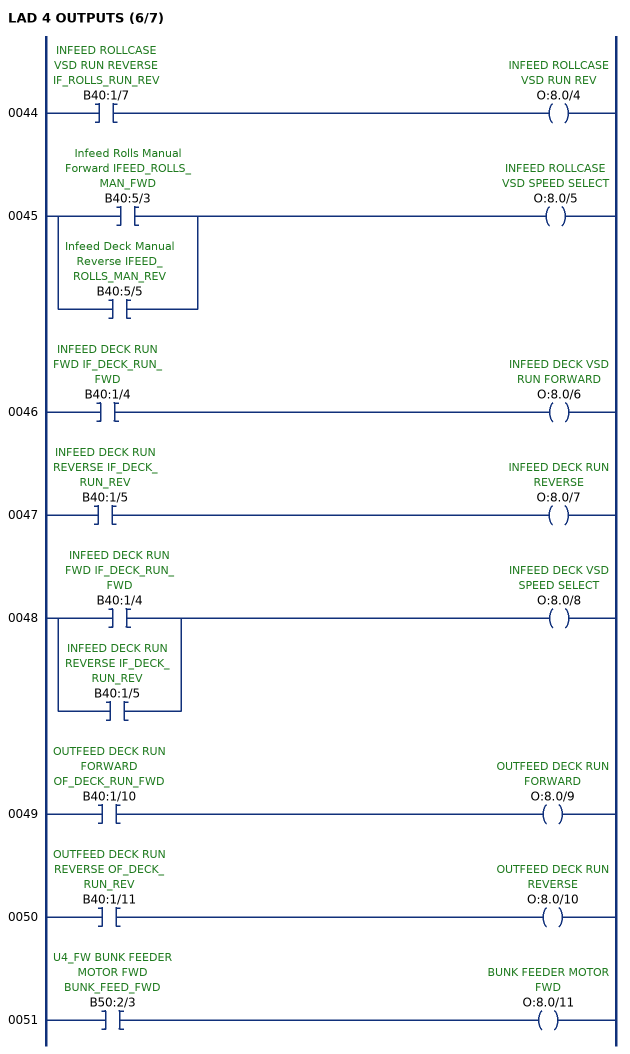
% Rung: 44 %
SOR XIC B40:1/7 OTE O:8.0/4 EOR
%   B40:1/7  IF_ROLLS_RUN_REV  "INFEED ROLLCASE VSD RUN REVERSE" %
%   O:8.0/4  "INFEED ROLLCASE VSD RUN REV" %
% Rung: 45 %
SOR BST XIC B40:5/3 NXB XIC B40:5/5 BND OTE O:8.0/5 EOR
%   B40:5/3  IFEED_ROLLS_MAN_FWD  "Infeed Rolls Manual Forward" %
%   B40:5/5  IFEED_ROLLS_MAN_REV  "Infeed Deck Manual Reverse" %
%   O:8.0/5  "INFEED ROLLCASE VSD SPEED SELECT" %
% Rung: 46 %
SOR XIC B40:1/4 OTE O:8.0/6 EOR
%   B40:1/4  IF_DECK_RUN_FWD  "INFEED DECK RUN FWD" %
%   O:8.0/6  "INFEED DECK VSD RUN FORWARD" %
% Rung: 47 %
SOR XIC B40:1/5 OTE O:8.0/7 EOR
%   B40:1/5  IF_DECK_RUN_REV  "INFEED DECK RUN REVERSE" %
%   O:8.0/7  "INFEED DECK RUN REVERSE" %
% Rung: 48 %
SOR BST XIC B40:1/4 NXB XIC B40:1/5 BND OTE O:8.0/8 EOR
%   B40:1/4  IF_DECK_RUN_FWD  "INFEED DECK RUN FWD" %
%   B40:1/5  IF_DECK_RUN_REV  "INFEED DECK RUN REVERSE" %
%   O:8.0/8  "INFEED DECK VSD SPEED SELECT" %
% Rung: 49 %
SOR XIC B40:1/10 OTE O:8.0/9 EOR
%   B40:1/10  OF_DECK_RUN_FWD  "OUTFEED DECK RUN FORWARD" %
%   O:8.0/9  "OUTFEED DECK RUN FORWARD" %
% Rung: 50 %
SOR XIC B40:1/11 OTE O:8.0/10 EOR
%   B40:1/11  OF_DECK_RUN_REV  "OUTFEED DECK RUN REVERSE" %
%   O:8.0/10  "OUTFEED DECK RUN REVERSE" %
% Rung: 51 %
SOR XIC B50:2/3 OTE O:8.0/11 EOR
%   B50:2/3  BUNK_FEED_FWD  "U4_FW BUNK FEEDER MOTOR FWD" %
%   O:8.0/11  "BUNK FEEDER MOTOR FWD" %

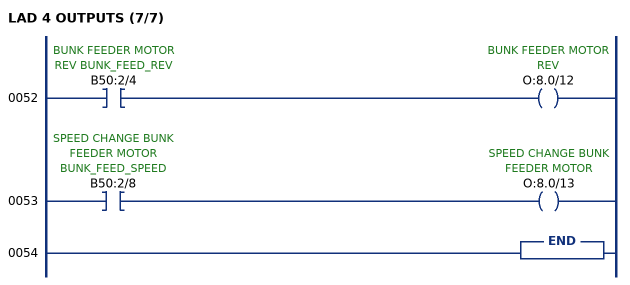
% Rung: 52 %
SOR XIC B50:2/4 OTE O:8.0/12 EOR
%   B50:2/4  BUNK_FEED_REV  "BUNK FEEDER MOTOR REV" %
%   O:8.0/12  "BUNK FEEDER MOTOR REV" %
% Rung: 53 %
SOR XIC B50:2/8 OTE O:8.0/13 EOR
%   B50:2/8  BUNK_FEED_SPEED  "SPEED CHANGE BUNK FEEDER MOTOR" %
%   O:8.0/13  "SPEED CHANGE BUNK FEEDER MOTOR" %
% Rung: 54 %
SOR END EOR

LADDER 5 "INTERF OP"
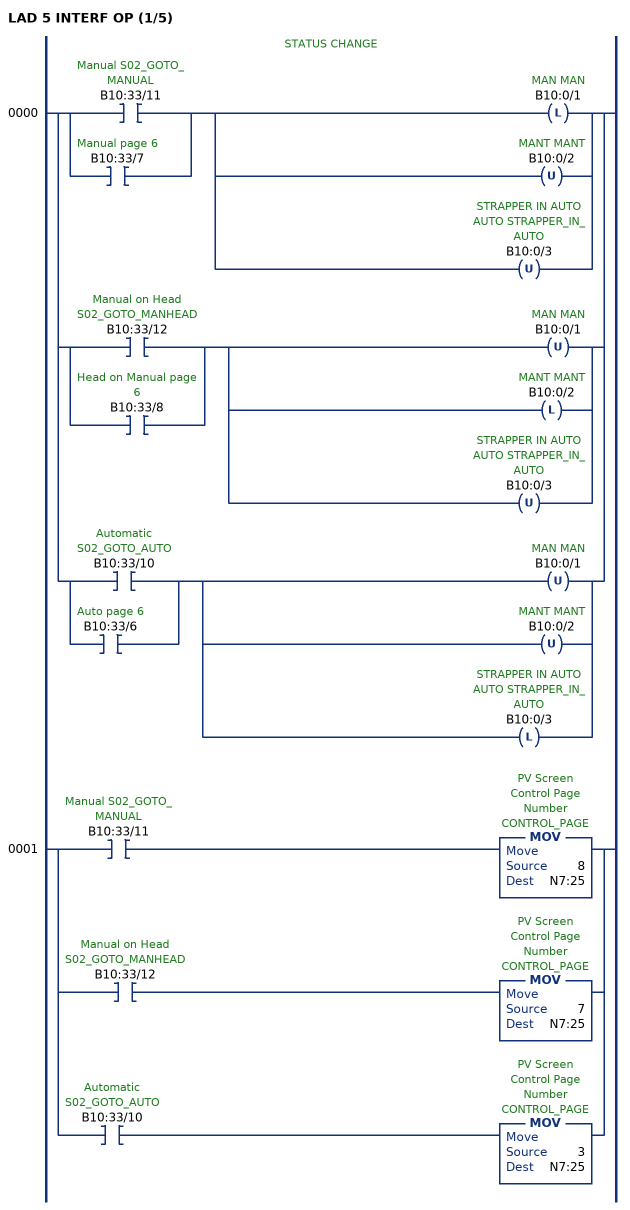
% Rung: 0 %
% STATUS CHANGE %
SOR BST BST XIC B10:33/11 NXB XIC B10:33/7 BND BST OTL B10:0/1 NXB BST OTU B10:0/2 NXB OTU B10:0/3 BND BND NXB BST BST XIC B10:33/12 NXB XIC B10:33/8 BND BST OTU B10:0/1 NXB BST OTL B10:0/2 NXB OTU B10:0/3 BND BND NXB BST XIC B10:33/10 NXB XIC B10:33/6 BND BST OTU B10:0/1 NXB BST OTU B10:0/2 NXB OTL B10:0/3 BND BND BND BND EOR
%   B10:33/11  S02_GOTO_MANUAL  "Manual" %
%   B10:33/7  "Manual page 6" %
%   B10:0/1  MAN  "MAN" %
%   B10:0/2  MANT  "MANT" %
%   B10:0/3  STRAPPER_IN_AUTO  "STRAPPER IN AUTO AUTO" %
%   B10:33/12  S02_GOTO_MANHEAD  "Manual on Head" %
%   B10:33/8  "Head on Manual page 6" %
%   B10:33/10  S02_GOTO_AUTO  "Automatic" %
%   B10:33/6  "Auto page 6" %
% Rung: 1 %
SOR BST XIC B10:33/11 MOV 8 N7:25 NXB BST XIC B10:33/12 MOV 7 N7:25 NXB XIC B10:33/10 MOV 3 N7:25 BND BND EOR
%   B10:33/11  S02_GOTO_MANUAL  "Manual" %
%   N7:25  CONTROL_PAGE  "PV Screen Control Page Number" %
%   B10:33/12  S02_GOTO_MANHEAD  "Manual on Head" %
%   B10:33/10  S02_GOTO_AUTO  "Automatic" %

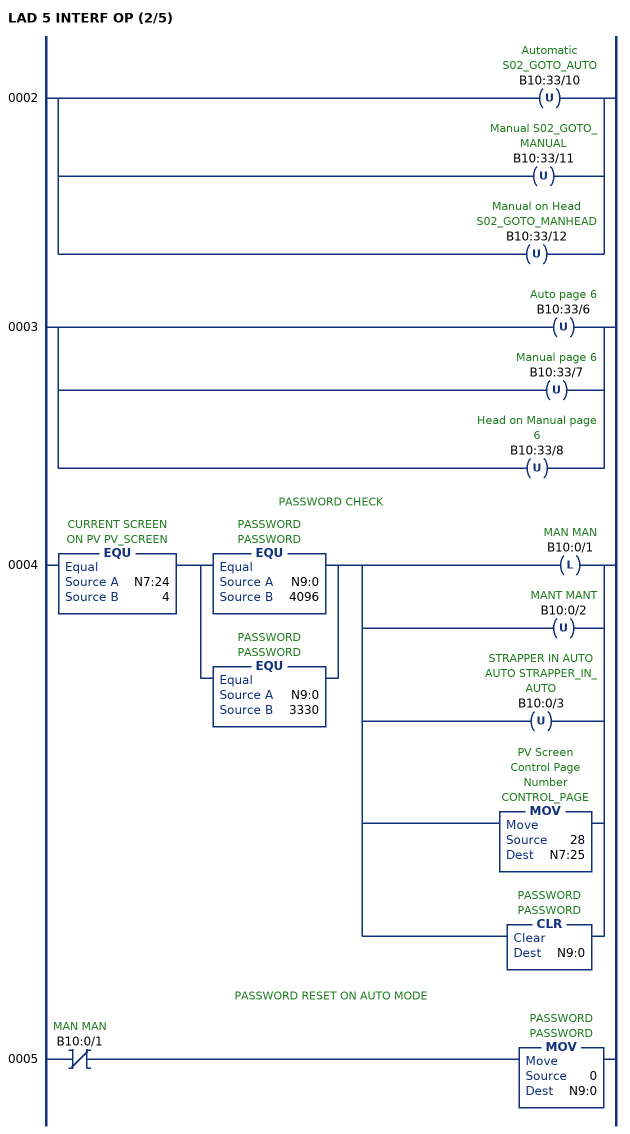
% Rung: 2 %
SOR BST OTU B10:33/10 NXB BST OTU B10:33/11 NXB OTU B10:33/12 BND BND EOR
%   B10:33/10  S02_GOTO_AUTO  "Automatic" %
%   B10:33/11  S02_GOTO_MANUAL  "Manual" %
%   B10:33/12  S02_GOTO_MANHEAD  "Manual on Head" %
% Rung: 3 %
SOR BST OTU B10:33/6 NXB BST OTU B10:33/7 NXB OTU B10:33/8 BND BND EOR
%   B10:33/6  "Auto page 6" %
%   B10:33/7  "Manual page 6" %
%   B10:33/8  "Head on Manual page 6" %
% Rung: 4 %
% PASSWORD CHECK %
SOR EQU N7:24 4 BST EQU N9:0 4096 NXB EQU N9:0 3330 BND BST BST BST OTL B10:0/1 NXB BST OTU B10:0/2 NXB OTU B10:0/3 BND BND NXB MOV 28 N7:25 BND NXB CLR N9:0 BND EOR
%   N7:24  PV_SCREEN  "CURRENT SCREEN ON PV" %
%   N9:0  PASSWORD  "PASSWORD" %
%   B10:0/1  MAN  "MAN" %
%   B10:0/2  MANT  "MANT" %
%   B10:0/3  STRAPPER_IN_AUTO  "STRAPPER IN AUTO AUTO" %
%   N7:25  CONTROL_PAGE  "PV Screen Control Page Number" %
% Rung: 5 %
% PASSWORD RESET ON AUTO MODE %
SOR XIO B10:0/1 MOV 0 N9:0 EOR
%   B10:0/1  MAN  "MAN" %
%   N9:0  PASSWORD  "PASSWORD" %

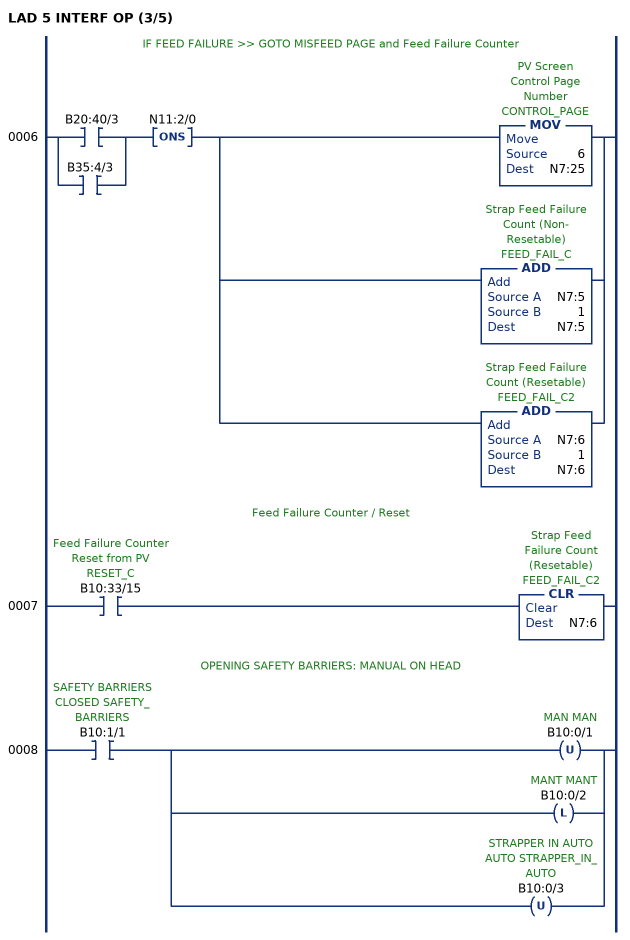
% Rung: 6 %
% IF FEED FAILURE >> GOTO MISFEED PAGE and Feed Failure Counter %
SOR BST XIC B20:40/3 NXB XIC B35:4/3 BND ONS N11:2/0 BST MOV 6 N7:25 NXB BST ADD N7:5 1 N7:5 NXB ADD N7:6 1 N7:6 BND BND EOR
%   N7:25  CONTROL_PAGE  "PV Screen Control Page Number" %
%   N7:5  FEED_FAIL_C  "Strap Feed Failure Count (Non-Resetable)" %
%   N7:6  FEED_FAIL_C2  "Strap Feed Failure Count (Resetable)" %
% Rung: 7 %
% Feed Failure Counter / Reset %
SOR XIC B10:33/15 CLR N7:6 EOR
%   B10:33/15  RESET_C  "Feed Failure Counter Reset from PV" %
%   N7:6  FEED_FAIL_C2  "Strap Feed Failure Count (Resetable)" %
% Rung: 8 %
% OPENING SAFETY BARRIERS: MANUAL ON HEAD %
SOR XIC B10:1/1 BST OTU B10:0/1 NXB BST OTL B10:0/2 NXB OTU B10:0/3 BND BND EOR
%   B10:1/1  SAFETY_BARRIERS  "SAFETY BARRIERS CLOSED" %
%   B10:0/1  MAN  "MAN" %
%   B10:0/2  MANT  "MANT" %
%   B10:0/3  STRAPPER_IN_AUTO  "STRAPPER IN AUTO AUTO" %

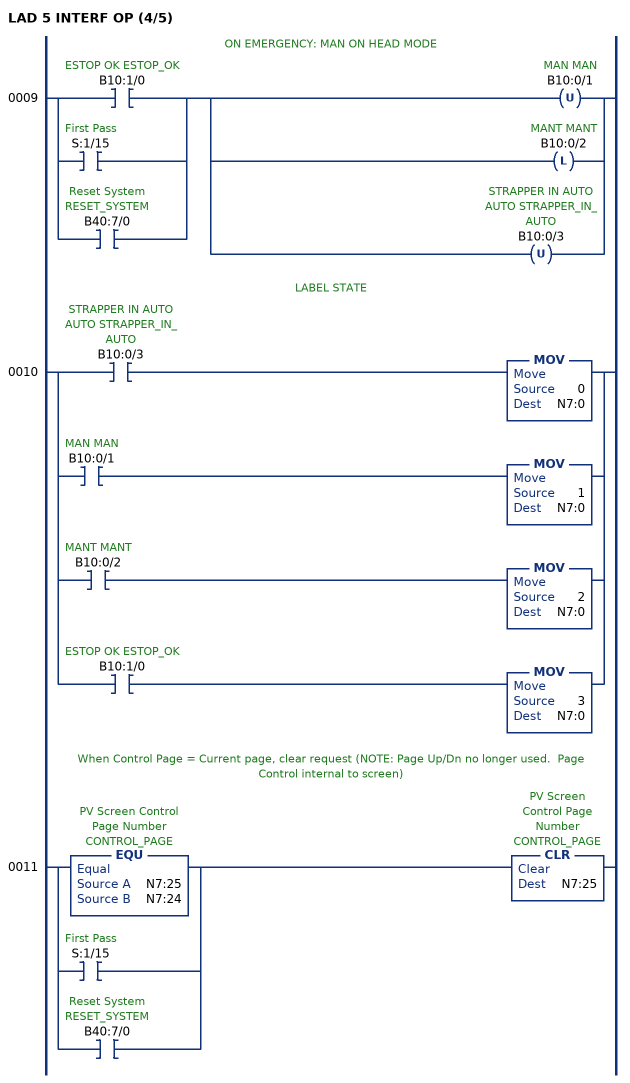
% Rung: 9 %
% ON EMERGENCY: MAN ON HEAD MODE %
SOR BST XIC B10:1/0 NXB XIC S:1/15 NXB XIC B40:7/0 BND BST OTU B10:0/1 NXB BST OTL B10:0/2 NXB OTU B10:0/3 BND BND EOR
%   B10:1/0  ESTOP_OK  "ESTOP OK" %
%   S:1/15  "First Pass" %
%   B40:7/0  RESET_SYSTEM  "Reset System" %
%   B10:0/1  MAN  "MAN" %
%   B10:0/2  MANT  "MANT" %
%   B10:0/3  STRAPPER_IN_AUTO  "STRAPPER IN AUTO AUTO" %
% Rung: 10 %
% LABEL STATE %
SOR BST XIC B10:0/3 MOV 0 N7:0 NXB BST XIC B10:0/1 MOV 1 N7:0 NXB BST XIC B10:0/2 MOV 2 N7:0 NXB XIC B10:1/0 MOV 3 N7:0 BND BND BND EOR
%   B10:0/3  STRAPPER_IN_AUTO  "STRAPPER IN AUTO AUTO" %
%   B10:0/1  MAN  "MAN" %
%   B10:0/2  MANT  "MANT" %
%   B10:1/0  ESTOP_OK  "ESTOP OK" %
% Rung: 11 %
% When Control Page = Current page, clear request (NOTE: Page Up/Dn no longer used.  Page Control internal to screen) %
SOR BST EQU N7:25 N7:24 NXB XIC S:1/15 NXB XIC B40:7/0 BND CLR N7:25 EOR
%   N7:25  CONTROL_PAGE  "PV Screen Control Page Number" %
%   N7:24  PV_SCREEN  "CURRENT SCREEN ON PV" %
%   S:1/15  "First Pass" %
%   B40:7/0  RESET_SYSTEM  "Reset System" %

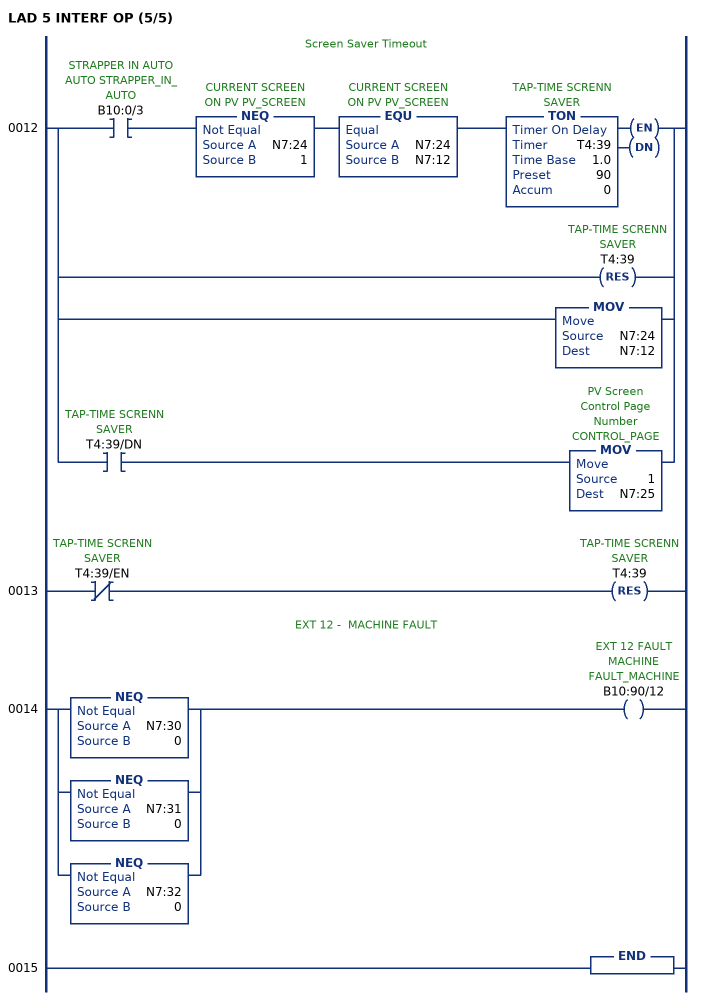
% Rung: 12 %
% Screen Saver Timeout %
SOR BST XIC B10:0/3 NEQ N7:24 1 EQU N7:24 N7:12 TON T4:39 1.0 90 0 NXB RES T4:39 NXB MOV N7:24 N7:12 NXB XIC T4:39/DN MOV 1 N7:25 BND EOR
%   B10:0/3  STRAPPER_IN_AUTO  "STRAPPER IN AUTO AUTO" %
%   N7:24  PV_SCREEN  "CURRENT SCREEN ON PV" %
%   T4:39  "TAP-TIME SCRENN SAVER" %
%   N7:25  CONTROL_PAGE  "PV Screen Control Page Number" %
% Rung: 13 %
SOR XIO T4:39/EN RES T4:39 EOR
%   T4:39  "TAP-TIME SCRENN SAVER" %
% Rung: 14 %
% EXT 12 -  MACHINE FAULT %
SOR BST NEQ N7:30 0 NXB BST NEQ N7:31 0 NXB NEQ N7:32 0 BND BND OTE B10:90/12 EOR
%   B10:90/12  FAULT_MACHINE  "EXT 12 FAULT MACHINE" %
% Rung: 15 %
SOR END EOR

LADDER 6 "COEFF."    % COEFFICIENT OF SEALING %
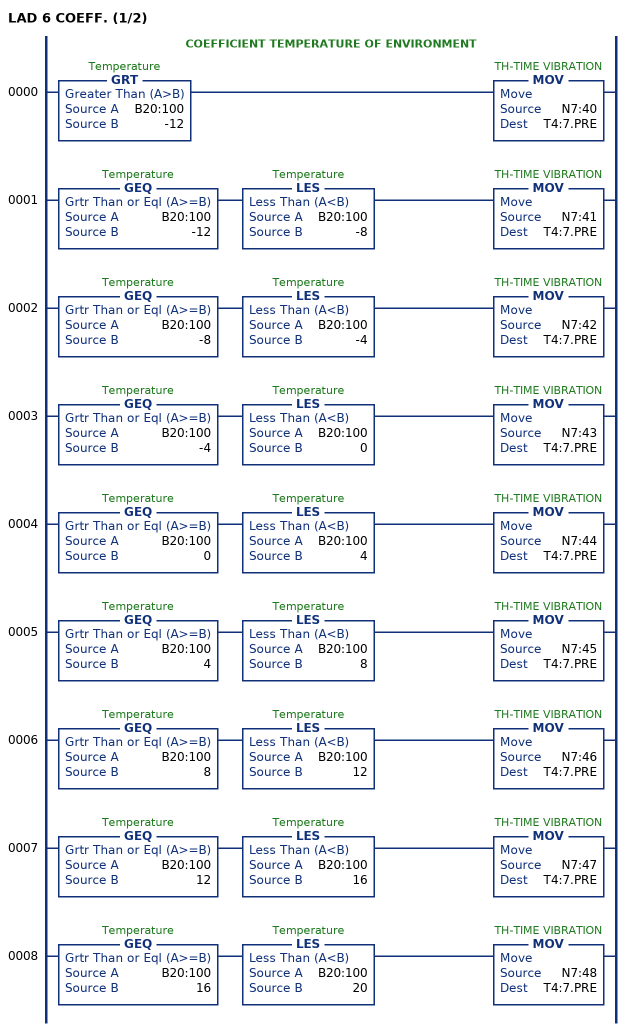
% Rung: 0 %
% TITLE: COEFFICIENT TEMPERATURE OF ENVIRONMENT %
SOR GRT B20:100 -12 MOV N7:40 T4:7.PRE EOR
%   B20:100  "Temperature" %
%   N7:40  "KA" %
%   T4:7  "TH-TIME VIBRATION" %
% Rung: 1 %
SOR GEQ B20:100 -12 LES B20:100 -8 MOV N7:41 T4:7.PRE EOR
%   B20:100  "Temperature" %
%   N7:41  "KB" %
%   T4:7  "TH-TIME VIBRATION" %
% Rung: 2 %
SOR GEQ B20:100 -8 LES B20:100 -4 MOV N7:42 T4:7.PRE EOR
%   B20:100  "Temperature" %
%   N7:42  "KC" %
%   T4:7  "TH-TIME VIBRATION" %
% Rung: 3 %
SOR GEQ B20:100 -4 LES B20:100 0 MOV N7:43 T4:7.PRE EOR
%   B20:100  "Temperature" %
%   N7:43  "KD" %
%   T4:7  "TH-TIME VIBRATION" %
% Rung: 4 %
SOR GEQ B20:100 0 LES B20:100 4 MOV N7:44 T4:7.PRE EOR
%   B20:100  "Temperature" %
%   N7:44  "KE" %
%   T4:7  "TH-TIME VIBRATION" %
% Rung: 5 %
SOR GEQ B20:100 4 LES B20:100 8 MOV N7:45 T4:7.PRE EOR
%   B20:100  "Temperature" %
%   N7:45  "KF" %
%   T4:7  "TH-TIME VIBRATION" %
% Rung: 6 %
SOR GEQ B20:100 8 LES B20:100 12 MOV N7:46 T4:7.PRE EOR
%   B20:100  "Temperature" %
%   N7:46  "KG" %
%   T4:7  "TH-TIME VIBRATION" %
% Rung: 7 %
SOR GEQ B20:100 12 LES B20:100 16 MOV N7:47 T4:7.PRE EOR
%   B20:100  "Temperature" %
%   N7:47  "KH" %
%   T4:7  "TH-TIME VIBRATION" %
% Rung: 8 %
SOR GEQ B20:100 16 LES B20:100 20 MOV N7:48 T4:7.PRE EOR
%   B20:100  "Temperature" %
%   N7:48  "KJ" %
%   T4:7  "TH-TIME VIBRATION" %

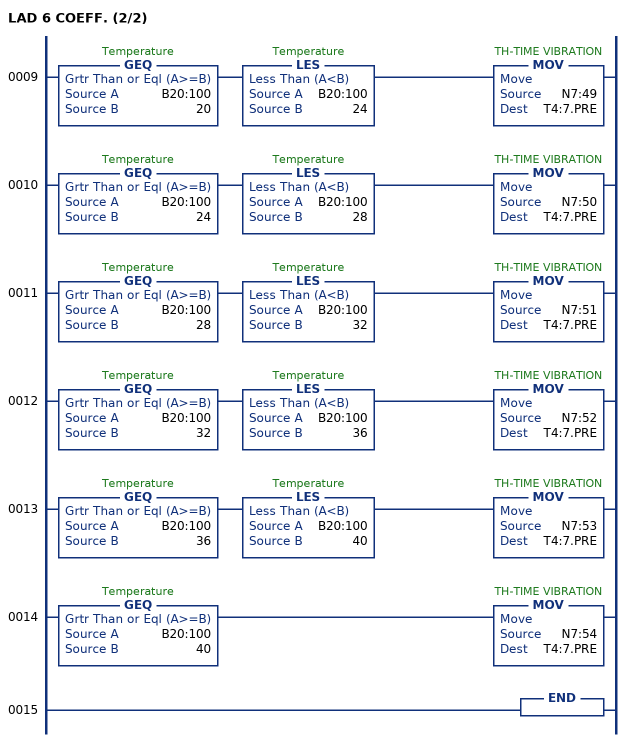
% Rung: 9 %
SOR GEQ B20:100 20 LES B20:100 24 MOV N7:49 T4:7.PRE EOR
%   B20:100  "Temperature" %
%   N7:49  "KK" %
%   T4:7  "TH-TIME VIBRATION" %
% Rung: 10 %
SOR GEQ B20:100 24 LES B20:100 28 MOV N7:50 T4:7.PRE EOR
%   B20:100  "Temperature" %
%   N7:50  "KL" %
%   T4:7  "TH-TIME VIBRATION" %
% Rung: 11 %
SOR GEQ B20:100 28 LES B20:100 32 MOV N7:51 T4:7.PRE EOR
%   B20:100  "Temperature" %
%   N7:51  "KM" %
%   T4:7  "TH-TIME VIBRATION" %
% Rung: 12 %
SOR GEQ B20:100 32 LES B20:100 36 MOV N7:52 T4:7.PRE EOR
%   B20:100  "Temperature" %
%   N7:52  "KN" %
%   T4:7  "TH-TIME VIBRATION" %
% Rung: 13 %
SOR GEQ B20:100 36 LES B20:100 40 MOV N7:53 T4:7.PRE EOR
%   B20:100  "Temperature" %
%   N7:53  "KO" %
%   T4:7  "TH-TIME VIBRATION" %
% Rung: 14 %
SOR GEQ B20:100 40 MOV N7:54 T4:7.PRE EOR
%   B20:100  "Temperature" %
%   N7:54  "KP" %
%   T4:7  "TH-TIME VIBRATION" %
% Rung: 15 %
SOR END EOR

LADDER 7 "DISPENSER"
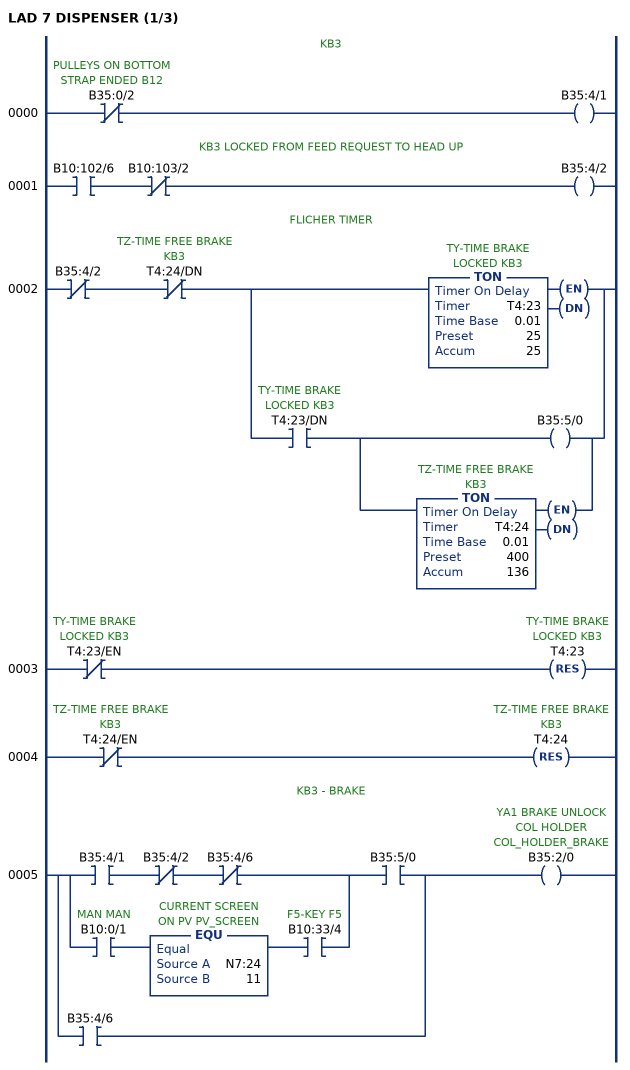
% Rung: 0 %
% KB3 %
SOR XIO B35:0/2 OTE B35:4/1 EOR
%   B35:0/2  B12  "PULLEYS ON BOTTOM STRAP ENDED" %
% Rung: 1 %
% KB3 LOCKED FROM FEED REQUEST TO HEAD UP %
SOR XIC B10:102/6 XIO B10:103/2 OTE B35:4/2 EOR
% Rung: 2 %
% FLICHER TIMER %
SOR XIO B35:4/2 XIO T4:24/DN BST TON T4:23 0.01 25 25 NXB XIC T4:23/DN BST OTE B35:5/0 NXB TON T4:24 0.01 400 136 BND BND EOR
%   T4:24  "TZ-TIME FREE BRAKE KB3" %
%   T4:23  "TY-TIME BRAKE LOCKED KB3" %
% Rung: 3 %
SOR XIO T4:23/EN RES T4:23 EOR
%   T4:23  "TY-TIME BRAKE LOCKED KB3" %
% Rung: 4 %
SOR XIO T4:24/EN RES T4:24 EOR
%   T4:24  "TZ-TIME FREE BRAKE KB3" %
% Rung: 5 %
% KB3 - BRAKE %
SOR BST BST XIC B35:4/1 XIO B35:4/2 XIO B35:4/6 NXB XIC B10:0/1 EQU N7:24 11 XIC B10:33/4 BND XIC B35:5/0 NXB XIC B35:4/6 BND OTE B35:2/0 EOR
%   B10:0/1  MAN  "MAN" %
%   N7:24  PV_SCREEN  "CURRENT SCREEN ON PV" %
%   B10:33/4  F5  "F5-KEY" %
%   B35:2/0  COL_HOLDER_BRAKE  "YA1 BRAKE UNLOCK COL HOLDER" %

